(* PLC project mtcs_tmc, Institute of Astronomy Onto 0.0.1 *)
(* stored: creationDateTime 2024-10-22T16:57:18.797943, modificationDateTime 2024-10-22T16:57:18.797943 *)

TYPE TmcTimingMode : (LOCAL_CLOCK := 0, PTP_IEEE_1588 := 1);
END_TYPE

TYPE TmcAxesErrors : (AXES_NO_ERROR := 0, AXES_OBJECT_RC_OUT_OF_RANGE := 1, AXES_OBJECT_DC_OUT_OF_RANGE := 2, AXES_OBJECT_PR_OUT_OF_RANGE := 3, AXES_OBJECT_PD_OUT_OF_RANGE := 4, AXES_OBJECT_PX_OUT_OF_RANGE := 5, AXES_EQ_OUT_OF_RANGE := 6, AXES_LOCATION_XP_OUT_OF_RANGE := 7, AXES_LOCATION_YP_OUT_OF_RANGE := 8, AXES_LOCATION_DX_OUT_OF_RANGE := 9, AXES_LOCATION_DY_OUT_OF_RANGE := 10, AXES_LOCATION_ELONG_OUT_OF_RANGE := 11, AXES_LOCATION_PHI_OUT_OF_RANGE := 12, AXES_LOCATION_HM_OUT_OF_RANGE := 13, AXES_LOCATION_TK_OUT_OF_RANGE := 14, AXES_LOCATION_PHPA_OUT_OF_RANGE := 15, AXES_LOCATION_RH_OUT_OF_RANGE := 16, AXES_LOCATION_WLFQ_OUT_OF_RANGE := 17, AXES_LOCATION_TLR_OUT_OF_RANGE := 18, AXES_FEEDBACK_AZ_OUT_OF_RANGE := 19, AXES_FEEDBACK_EL_OUT_OF_RANGE := 20);
END_TYPE

TYPE TmcTimingErrors : (TIMING_NO_ERROR := 0, TIMING_DUT_OUT_OF_RANGE := 1, TIMING_GETCURDCTIME_FAILED := 2);
END_TYPE

TYPE TmcTarget : STRUCT
  rc : LREAL;  (* Object mean right ascention (alpha) in radians *)
  dc : LREAL;  (* Object mean declination (delta) in radians *)
  pr : INT;  (* Object Right Ascention proper motion in radians/year (do not multiply by cos(dc)!) *)
  pd : INT;  (* Object declination proper motion in radians/year *)
  px : LREAL;  (* Object parallax in arcseconds *)
  rv : LREAL;  (* Object radial velocity in km/s *)
END_STRUCT;
END_TYPE

TYPE TmcLocation : STRUCT
  xp : REAL;  (* Earth polar motion x in radians *)
  yp : REAL;  (* Earth polar motion y in radians *)
  dx : REAL;  (* Nutation adjustment dX in radians *)
  dy : REAL;  (* Nutation adjustment dY in radians *)
  elong : LREAL;  (* East longitude in radians *)
  phi : LREAL;  (* latitude in radians *)
  hm : REAL;  (* Height above sea level in meters *)
  tk : REAL;  (* Local temperature in Kelvin *)
  phpa : REAL;  (* Local pressure in hectoPascal = millibar *)
  rh : REAL;  (* Local relative humidity as a fraction (0...1) *)
  wlfq : REAL;  (* Observing wavelength in microns *)
  tlr : REAL;  (* Tropospheric lapse rate in K/m *)
END_STRUCT;
END_TYPE

TYPE TmcAzEl : STRUCT
  az : LREAL;  (* Azimuth in radians *)
  el : LREAL;  (* Elevation in radians *)
END_STRUCT;
END_TYPE

TYPE TmcAzElFull : STRUCT
  az : LREAL;  (* Azimuth in radians *)
  azd : LREAL;  (* Azimuth velocity in radians per second *)
  azdd : LREAL;  (* Azimuth acceleration in radians/s2 *)
  el : LREAL;  (* Elevation in radians *)
  eld : LREAL;  (* Elevation velocity in radians per second *)
  eldd : LREAL;  (* Elevation acceleration in radians/s2 *)
  pa : LREAL;  (* Parallactic Angle in radians *)
  pad : LREAL;  (* Parallactic Angle velocity in radians per second *)
  padd : LREAL;  (* Parallactic Angle acceleration in radians/s2 *)
END_STRUCT;
END_TYPE

TYPE TmcRaDec : STRUCT
  ra : LREAL;  (* Right ascention (alpha) in radians *)
  dec : LREAL;  (* Declination (delta) in radians *)
END_STRUCT;
END_TYPE

TYPE TmcObserved : STRUCT
  aob : LREAL;  (* Observed azimuth (radians: North=0, East=PI/2) *)
  zob : LREAL;  (* Observed zentih distance (radians) *)
  hob : LREAL;  (* Observed hour angle (radians) *)
  dob : LREAL;  (* Observed declination (radians) *)
  rob : LREAL;  (* Observed right ascention (radians) *)
END_STRUCT;
END_TYPE

TYPE TmcTrue : STRUCT
  elong : LREAL;  (* True longitude of the site (radians, east +ve) *)
  phi : LREAL;  (* True geodetic latitude of the site (radians) *)
  daz : LREAL;  (* Azimuth correction for true longitude and latitude (terrestrial - celestial, radians) *)
END_STRUCT;
END_TYPE

TYPE TmcProcessedTarget : STRUCT
  given : TmcTarget;  (* The originally given target *)
  apparent : TmcRaDec;  (* Apparent target position *)
  quick : TmcAzElFull;  (* Quick computation results of target (without atmospheric refraction) *)
  observed : TmcObserved;  (* Observed target position *)
  observedFull : TmcAzElFull;  (* Observed target position/velocity/acceleration *)
  isValid : BOOL;  (* Is the target valid? *)
  isTooLow : BOOL;  (* Is the target too low? *)
END_STRUCT;
END_TYPE

TYPE TmcProcessedFeedback : STRUCT
  apparent : TmcRaDec;  (* Apparent feedback position *)
  mean : TmcRaDec;  (* Mean feedback position *)
  isValid : BOOL;  (* Is the feedback valid? *)
  isTooLow : BOOL;  (* Is the feedback too low? *)
END_STRUCT;
END_TYPE

TYPE TmcDateTime : STRUCT
  years : DINT;  (* Years, e.g. 2016 *)
  months : DINT;  (* Months, [1..12] *)
  days : DINT;  (* Days, [1..31] *)
  hours : DINT;  (* Hours, [0..23] *)
  minutes : DINT;  (* Minutes, [0..59] *)
  seconds : DINT;  (* Secconds, [0..60] (60 during leap second event!) *)
  microseconds : DINT;  (* Microseconds, [0..999999] *)
  fractionOfDay : LREAL;  (* Fraction of the day, [0.0..1.0[ *)
END_STRUCT;
END_TYPE

TYPE TmcUnixTime : STRUCT
  sec : LINT;  (* Seconds from Jan 1, 1970 *)
  usec : LINT;  (* Microseconds *)
END_STRUCT;
END_TYPE

TYPE TmcUtcTime : STRUCT
  dcTime : LINT;  (* DC time *)
  mode : TmcTimingMode;  (* Local clock or PTP? *)
  unixTime : TmcUnixTime;  (* UTC as Unix time *)
  mjd : LREAL;  (* UTC as Modified Julian Days *)
  dateTime : TmcDateTime;  (* EtherCAT master: Offset between DC and TwinCAT time (in ns) *)
END_STRUCT;
END_TYPE

TYPE TmcUt1Time : STRUCT
  mjd : LREAL;  (* UT1 as Modified Julian Days *)
END_STRUCT;
END_TYPE

TYPE TmcFromIoEcatMaster : STRUCT
  dcToTcTimeOffset : LINT;  (* EtherCAT master: Offset between DC and TwinCAT time (in ns) *)
  dcToExtTimeOffset : LINT;  (* EtherCAT master: Offset between Dc and external time (in ns) *)
END_STRUCT;
END_TYPE

TYPE TmcFromIoEL6688 : STRUCT
  internalTimestamp : ULINT;  (* EL6688 module: internal timestamp *)
  externalTimestamp : ULINT;  (* EL6688 module: external timestamp *)
  notConnected : BOOL;  (* EL6688 module: not connected *)
  updateToggle : BOOL;  (* EL6688 module: update toggle *)
END_STRUCT;
END_TYPE

TYPE TmcFromIo : STRUCT
  fromEL6688 : TmcFromIoEL6688;  (* Connect to inputs of EL6688 *)
  fromEcatMaster : TmcFromIoEcatMaster;  (* Connect to inputs of EtherCAT master *)
END_STRUCT;
END_TYPE

TYPE TmcFromPlcAxes : STRUCT
  object : TmcTarget;  (* Target *)
  equinox : LREAL;  (* Epoch of mean equinoxes (e.g. 2000.0) *)
  location : TmcLocation;  (* Location of the observatory *)
  feedback : TmcAzEl;  (* Feedback position (by the encoders) *)
END_STRUCT;
END_TYPE

TYPE TmcFromPlcTiming : STRUCT
  dut : LREAL;  (* Delta UT (=UT1 - UTC, floating point between 0 and 1 second) *)
  leapSeconds : DINT;  (* Number of leap seconds *)
  alwaysUseLocalClock : BOOL;  (* If TRUE, then the local clock (source=LOCAL_CLOCK) will be used even if an external (more accurate!) clock is available *)
END_STRUCT;
END_TYPE

TYPE TmcFromPlc : STRUCT
  fromAxes : TmcFromPlcAxes;  (* Connect to outputs of PLC - MTCS - Axes *)
  fromTiming : TmcFromPlcTiming;  (* Connect to outputs of PLC - MTCS - Services/Timing *)
END_STRUCT;
END_TYPE

TYPE TmcToPlcAxes : STRUCT
  polmo : TmcTrue;  (* True longitude/latitude/azimuth after polar motion correction *)
  last : LREAL;  (* Local apparent sidereal time *)
  ha : LREAL;  (* Hour angle in radians *)
  object : TmcProcessedTarget;  (* Processed target *)
  feedback : TmcProcessedFeedback;  (* Processed feedback *)
  error : TmcAxesErrors;  (* 0 = no error *)
END_STRUCT;
END_TYPE

TYPE TmcToPlcTiming : STRUCT
  utc : TmcUtcTime;  (* UTC time *)
  ut1 : TmcUt1Time;  (* UT1 time *)
  error : TmcTimingErrors;  (* 0 = no error *)
END_STRUCT;
END_TYPE

TYPE TmcToPlc : STRUCT
  toAxes : TmcToPlcAxes;  (* Connect to inputs of PLC - MTCS - Axes *)
  toTiming : TmcToPlcTiming;  (* Connect to inputs of PLC - MTCS - Services/Timing *)
END_STRUCT;
END_TYPE
